Staubli VAL3: HerePoint.pgx

public program HerePoint(num x_nIndex)
  local tool l_tTool
  local point l_pHere
  local frame l_fFrame
  local num i
  local num l_nIndex
  local num l_nSize
  local string l_sMessage
begin
  //
  // take the point
  //
  // frame
  call getFrame(fSetFrame,false)
  // tool
  call tcp:getTool(l_tTool,pEditPoint.nIndexTool)
  // here
  l_pHere=here(l_tTool,fSetFrame)
  resetMotion()
  // check the index
  if pEditPoint.tData[x_nIndex].nType==1
    // save the trsf
    pEditPoint.tData[x_nIndex].pPoint.trsf=l_pHere.trsf
  else
    // search for the index of the point
    call getSizeItem(false,l_nSize)
    for i=0 to l_nSize-1
      if pEditPoint.tData[i].nType==1
        // save and exit
        l_nIndex=i
        i=l_nSize
      endIf
    endFor
    if pEditPoint.tData[l_nIndex].pPoint.trsf!={0,0,0,0,0,0}
      // compute the approch
      pEditPoint.tData[x_nIndex].pPoint.trsf=!pEditPoint.tData[l_nIndex].pPoint.trsf*l_pHere.trsf
    else
      // point not taught
      call language:message(l_sMessage,147)
      popUpMsg(l_sMessage)
    endIf
  endIf
  // check the moveType to save the config
  if pEditPoint.tData[x_nIndex].tSuper.moveType==0
    pEditPoint.tData[x_nIndex].pPoint.config=l_pHere.config
  else
    pEditPoint.tData[x_nIndex].pPoint.config={ssame,esame,wfree}
  endIf
  // to be save

end
